FUNCTION_BLOCK FB_Module_CoilHolder IMPLEMENTS I_Module
VAR_INPUT
	sName			: STRING[50];
	tTimeout		: TIME := T#0S;
END_VAR

VAR_IN_OUT
END_VAR

VAR_OUTPUT
	bEnabled     	: BOOL;
	eState			: E_State := E_State.DISABLED;
	eNextState		: E_State := E_State.DISABLED;
	nCurrentIndex	: INT;
	sStatusText 	: STRING[100];
END_VAR

VAR
	eLastState		: E_State;
	tTimeoutTimer	: TON;
	Components		: ARRAY [0..7] OF I_Component;

	fbMotor			: FB_Component_ACmotor;
	fbPistonLock	: FB_Component_SingleValveGuarded;	
	fbIndexReadyBit	: FB_Component_InductiveSensor;
	fbIndexBit1		: FB_Component_InductiveSensor;
	fbIndexBit2		: FB_Component_InductiveSensor;
	fbIndexBit3		: FB_Component_InductiveSensor;
	fbIndexBit4		: FB_Component_InductiveSensor;
	fbIndexBit5		: FB_Component_InductiveSensor;
	
	nTargetIndex	: INT;
	cwSteps			: INT;
	ccwSteps		: INT;
	shortestDistance: INT;
END_VAR

VAR CONSTANT
	DISABLED		: E_State := E_State.DISABLED;
	READY			: E_State := E_State.READY;
	BUSY			: E_State := E_State.BUSY;
	HALTED			: E_State := E_State.HALTED;
	TIMEOUT			: E_State := E_State.TIMEOUT;
	
	CW				: E_RotationDirection := E_RotationDirection.CW;
	CCW				: E_RotationDirection := E_RotationDirection.CCW;
	
	FOFF			: E_LenzeJogFreq := E_LenzeJogFreq.FOFF;
	F1				: E_LenzeJogFreq := E_LenzeJogFreq.F1;
	F2				: E_LenzeJogFreq := E_LenzeJogFreq.F2;
	F3				: E_LenzeJogFreq := E_LenzeJogFreq.F3;
END_VAR

tTimeoutTimer(PT := tTimeout);

fbMotor(		sName := 'motor for coil holder', 
				bDeviceActive 	:= GVL.bLenze1Relay, 
				bE1jog1 		:= GVL.bLenze1JogBit1, 
				bE2jog2 		:= GVL.bLenze1JogBit2, 
				bE3DCbrake 		:= GVL.bLenze1InjectionBrake, 
				eE4Direction	:= gvl.bLenze1Direction);
				
fbPistonLock(	sName := 'lock for coil holder',
				bSensExtended := GVL.bCoilHolderUnlocked,
				bSensRetracted := GVL.bCoilHolderLocked,
				bOutput := GVL.bUnlockCoilHolder);

fbIndexReadyBit(sName := 'index ready bit for coil holder', bRawSignal := GVL.bCoilHolderIndexReady);

fbIndexBit1(sName := 'index bit 1 for coil holder', bRawSignal := GVL.bCoilHolderIndexBit1);
fbIndexBit2(sName := 'index bit 2 for coil holder', bRawSignal := GVL.bCoilHolderIndexBit2);
fbIndexBit3(sName := 'index bit 3 for coil holder', bRawSignal := GVL.bCoilHolderIndexBit3);
fbIndexBit4(sName := 'index bit 4 for coil holder', bRawSignal := GVL.bCoilHolderIndexBit4);
fbIndexBit5(sName := 'index bit 5 for coil holder', bRawSignal := GVL.bCoilHolderIndexBit5);

Components[0] := fbMotor;
Components[1] := fbPistonLock;
Components[2] := fbIndexReadyBit; 
Components[3] := fbIndexBit1; 
Components[4] := fbIndexBit2; 
Components[5] := fbIndexBit3; 
Components[6] := fbIndexBit4; 
Components[7] := fbIndexBit5; 

IF fbIndexReadyBit.bSensorActive THEN
	nCurrentIndex := 	TO_INT(	SHL(TO_UINT(fbIndexBit5.bSensorActive), 4) OR
								SHL(TO_UINT(fbIndexBit4.bSensorActive), 3) OR
								SHL(TO_UINT(fbIndexBit3.bSensorActive), 2) OR
								SHL(TO_UINT(fbIndexBit2.bSensorActive), 1) OR
						   		   (TO_UINT(fbIndexBit1.bSensorActive)));
END_IF

CASE eState OF
	DISABLED: 	sStatusText := 'Coil holder disabled';
	READY: 		sStatusText := CONCAT('coil holder is ready to operate and at index: ', INT_TO_STRING(nCurrentIndex));
	
	BUSY: 		IF fbPistonLock.bIsExtended THEN
					IF nTargetIndex = nCurrentIndex THEN
						fbMotor.M_SetFreq(Frequency := FOFF);
						fbPistonLock.M_Retract();
						eNextState := TIMEOUT;
					ELSE
						cwSteps  := (nTargetIndex - nCurrentIndex + 24) MOD 24;
						ccwSteps := (nCurrentIndex - nTargetIndex + 24) MOD 24;
						
						IF cwSteps <= ccwSteps THEN
							fbMotor.M_SetDir(Direction := CW);
							shortestDistance := cwSteps;
						ELSE
							fbMotor.M_SetDir(Direction := CCW);	
							shortestDistance := ccwSteps;
						END_IF
						
						IF nCurrentIndex <> nTargetIndex THEN
							IF shortestDistance <= 1 THEN
								fbMotor.M_SetFreq(Frequency := F1);	
							ELSIF shortestDistance <= 2 THEN
								fbMotor.M_SetFreq(Frequency := F2);
							ELSE
								fbMotor.M_SetFreq(Frequency := F3);
							END_IF
						ELSE
							fbMotor.M_SetFreq(Frequency := FOFF);
							fbPistonLock.M_Retract();
							eNextState := TIMEOUT;
						END_IF
					END_IF
				ELSE
					fbPistonLock.M_Extend();
				END_IF
	TIMEOUT:	sStatusText := 'Coil holder is in timeout';
				tTimeoutTimer(IN := TRUE);
				
				IF tTimeoutTimer.Q THEN
					tTimeoutTimer(IN := FALSE);
					eNextState := READY;
				END_IF
	HALTED:		sStatusText := 'Coil holder halted';
END_CASE 
eState := eNextState;

{warning 'add method implementation '}
METHOD M_Disable : BOOL

VAR
	idx: INT;
END_VAR
IF eState = READY THEN
	bEnabled	:= FALSE;
	eNextState	:= DISABLED;
	
	FOR idx := 0 TO 7 DO
    	Components[idx].M_Disable();
	END_FOR;
END_IF
END_METHOD

{warning 'add method implementation '}
METHOD M_Enable : BOOL

VAR
	idx: INT;
END_VAR
IF eState = DISABLED THEN
	bEnabled	:= TRUE;
	eNextState	:= READY;
	
	FOR idx := 0 TO 7 DO
    	Components[idx].M_Enable();
	END_FOR;
END_IF
END_METHOD

{warning 'add method implementation '}
METHOD M_Halt : BOOL

VAR
	idx: INT;
END_VAR
IF eState <> HALTED AND eState <> DISABLED THEN
	eLastState 		:= eState;
	eNextState		:= HALTED;
	FOR idx := 0 TO 7 DO
		Components[idx].M_Halt();
	END_FOR;
END_IF
END_METHOD

{warning 'add method implementation '}
METHOD M_Resume : BOOL

VAR
	idx: INT;
END_VAR
IF eState = HALTED THEN
	eNextState := eLastState;
	FOR idx := 0 TO 7 DO
		Components[idx].M_Resume();
	END_FOR;
END_IF
END_METHOD

METHOD M_SetTargetIndex : BOOL
VAR_INPUT
	index : INT;
END_VAR
IF eState = READY OR eState = BUSY THEN
	nTargetIndex 	:= index;
	eNextState 		:= BUSY;
END_IF
END_METHOD

END_FUNCTION_BLOCK

(* stored: Version 1.1.0.1, ProductVersion 3.1.4024.15
   POU FB_Module_CoilHolder: Id {fd1b5399-37e5-487f-bdd5-3dab864f6892}, SpecialFunc None
   Method M_Disable: Id {31e718ad-ecf7-45b5-a41a-22eaeff727dd}
   Method M_Enable: Id {475fe07d-e270-4d44-8ec8-53e8b17176f7}
   Method M_Halt: Id {d7178821-85b2-410c-991f-3a4798f76730}
   Method M_Resume: Id {8dc7de34-88d6-4b0d-8f3c-bb66d6524524}
   Method M_SetTargetIndex: Id {22a02a63-9ca4-4c51-89d8-9ddcfc4d1354} *)
